// TIA Portal V17 export
// export: Created 2023-05-07T12:12:23.8923214Z, ExportSetting WithDefaults, DisplayName Totally Integrated Automation Portal, DisplayVersion V17, DisplayName TIA Portal Openness, DisplayVersion V17, DisplayName TIA Portal Version Control Interface, DisplayVersion V17, DisplayName TIA Portal Test Suite Advanced, DisplayVersion V17, DisplayName STEP 7 Professional, DisplayVersion V17, DisplayName SIMATIC Energy Suite, DisplayVersion V17, DisplayName STEP 7 Safety, DisplayVersion V17, DisplayName WinCC Professional, DisplayVersion V17
DATA_BLOCK "Training_DB"   // DB10
VERSION : 0.1
// stored: AutoNumber true, InstanceOfName Training, InstanceOfType FB
"Training"
   // VAR_INPUT
   //    error_stop_m : Real;
   //    error_stop_i : Real;
   //    epoch_stop_m : Real;
   //    epoch_stop_i : Real;
   //    training_m : Bool;
   //    training_i : Bool;
   // END_VAR
   // VAR_OUTPUT
   //    error_ep_m { ExternalAccessible := 'False'; ExternalVisible := 'False'; ExternalWritable := 'False'} : Real;
   //    error_ep_i : Real;
   //    stop_m : Bool;
   //    stop_i : Bool;
   // END_VAR
   // VAR_IN_OUT
   //    epoch : Real;
   // END_VAR
   // VAR
   //    i : Int;
   //    long : Int;
   //    s : Array[0..7] of Real;
   //    o : Array[0..7] of Real;
   //    s2 : Real;
   //    e2 : Real;
   //    "e" : Array[0..7] of Real;
   //    x_m : Array[0..5] of Real;
   //    x_i : Array[0..5] of Real;
   //    n_m : Real;
   //    n_i : Real;
   // END_VAR
BEGIN
END_DATA_BLOCK
